(* CoDeSys 2.3.9.41 project: A1.pro *)
(* Libraries: STANDARD.LIB 15.6.21 11:37:35, IECSFC.LIB 15.6.21 11:37:35, SYSLIBTIME.LIB 18.6.21 10:30:26, SYSTASKINFO.LIB 18.6.21 10:30:26, ANALYZATION.LIB 15.6.21 11:37:35, SYSLIBCALLBACK.LIB 18.6.21 10:30:26 *)

(* PLC configuration (modules and I/O channels)
DI_1 AT %IX0.0 [BitInput] Discrete input 1 {ChannellName = Enter name}
DI_2 AT %IX0.1 [BitInput] Discrete input 2 {ChannellName = Enter name}
Discrete inputs [ID130] node 1, in %IB1 out %QB1 {ChannellName = Discrete inputs; Filtrationtime_GeneralINP = 16; PinCount = 16}
  AT %IB1.0 [ByteInput] 8 discrete inputs {ChannellName = Enter name}
  AT %IB1.1 [ByteInput] 8 discrete inputs {ChannellName = Enter name}
DO_1 AT %QX2.0 [BitOutput] Fast discrete output 1 {ChannellName = Enter name}
DO_2 AT %QX2.1 [BitOutput] Fast discrete output 2 {ChannellName = Enter name}
DO_3 AT %QX2.2 [BitOutput] Fast discrete output 3 {ChannellName = Enter name}
DO_4 AT %QX2.3 [BitOutput] Fast discrete output 4 {ChannellName = Enter name}
AT %QB3.0 [ByteOutput] 8 discrete outputs {ChannellName = Enter name}
AT %QB3.1 [ByteOutput] 8 discrete outputs {ChannellName = Enter name}
Special input [ID103] node 4, in %IB4 out %QB4 {ChannellName = Special input}
  AT %IX4.0 [BitInput] Special input {ChannellName = Enter name}
Special output [ID104] node 5, in %IB5 out %QB5 {ChannellName = Special output}
  AT %QX5.0 [BitOutput] Special output {ChannellName = Enter name}
RS-485-1 [COM1_USART] node 0, in %IB6.0.0 out %QB6.0.0 {ChannellName = RS-485-1; CommunicationSpeed = 115200; Parity = NO PARITY CHECK; BitLength = 8 bits; StopLength = One stop bit; InterfaceType = RS485; FrameOriented = RTU; Timeout = 0; Visibility = No}
2 byte [Register] node 1, in %IB6.1 out %QB6.1 {ChannellName = 2 byte}
  DI AT %QW6.1.0 [WordOutput] {ChannellName = Enter name}
2 byte [Register] node 2, in %IB6.2 out %QB6.2 {ChannellName = 2 byte}
  DOMod AT %QW6.2.0 [WordOutput] {ChannellName = Enter name}
2 byte [Register] node 3, in %IB6.3 out %QB6.3 {ChannellName = 2 byte}
  iPressure1 AT %QW6.3.0 [WordOutput] {ChannellName = Enter name}
2 byte [Register] node 4, in %IB6.4 out %QB6.4 {ChannellName = 2 byte}
  iPressure2 AT %QW6.4.0 [WordOutput] {ChannellName = Enter name}
2 byte [Register] node 5, in %IB6.5 out %QB6.5 {ChannellName = 2 byte}
  iPressure3 AT %QW6.5.0 [WordOutput] {ChannellName = Enter name}
2 byte [Register] node 6, in %IB6.6 out %QB6.6 {ChannellName = 2 byte}
  iPressure4 AT %QW6.6.0 [WordOutput] {ChannellName = Enter name}
2 byte [Register] node 7, in %IB6.7 out %QB6.7 {ChannellName = 2 byte}
  iPressure5 AT %QW6.7.0 [WordOutput] {ChannellName = Enter name}
2 byte [Register] node 8, in %IB6.8 out %QB6.8 {ChannellName = 2 byte}
  iPressure6 AT %QW6.8.0 [WordOutput] {ChannellName = Enter name}
2 byte [Register] node 9, in %IB6.9 out %QB6.9 {ChannellName = 2 byte}
  iPressureAll AT %QW6.9.0 [WordOutput] {ChannellName = Enter name}
2 byte [Register] node 10, in %IB6.10 out %QB6.10 {ChannellName = 2 byte}
  iPressureOil AT %QW6.10.0 [WordOutput] {ChannellName = Enter name}
2 byte [Register] node 11, in %IB6.11 out %QB6.11 {ChannellName = 2 byte}
  qNeedTemp AT %QW6.11.0 [WordOutput] {ChannellName = Enter name}
2 byte [Register] node 12, in %IB6.12 out %QB6.12 {ChannellName = 2 byte}
  qTempDelta AT %QW6.12.0 [WordOutput] {ChannellName = Enter name}
2 byte [Register] node 13, in %IB6.13 out %QB6.13 {ChannellName = 2 byte}
  qPressureOilMax AT %QW6.13.0 [WordOutput] {ChannellName = Enter name}
2 byte [Register] node 14, in %IB6.14 out %QB6.14 {ChannellName = 2 byte}
  qPressureMax AT %QW6.14.0 [WordOutput] {ChannellName = Enter name}
2 byte [Register] node 15, in %IB6.15 out %QB6.15 {ChannellName = 2 byte}
  qTempMin AT %QW6.15.0 [WordOutput] {ChannellName = Enter name}
2 byte [Register] node 16, in %IB6.16 out %QB6.16 {ChannellName = 2 byte}
  iAlarms AT %QW6.16.0 [WordOutput] {ChannellName = Enter name}
2 byte [Register] node 17, in %IB6.17 out %QB6.17 {ChannellName = 2 byte}
  qNeedPressure1 AT %QW6.17.0 [WordOutput] {ChannellName = Enter name}
2 byte [Register] node 18, in %IB6.18 out %QB6.18 {ChannellName = 2 byte}
  qNeedPressure2 AT %QW6.18.0 [WordOutput] {ChannellName = Enter name}
2 byte [Register] node 19, in %IB6.19 out %QB6.19 {ChannellName = 2 byte}
  qNeedPressure3 AT %QW6.19.0 [WordOutput] {ChannellName = Enter name}
2 byte [Register] node 20, in %IB6.20 out %QB6.20 {ChannellName = 2 byte}
  qNeedPressure4 AT %QW6.20.0 [WordOutput] {ChannellName = Enter name}
  qNeedPressure5 AT %QW6.21.0 [WordOutput] {ChannellName = Enter name}
  qNeedPressure6 AT %QW6.22.0 [WordOutput] {ChannellName = Enter name}
  iTemp1 AT %QW6.23.0 [WordOutput] {ChannellName = Enter name}
  iTemp2 AT %QW6.24.0 [WordOutput] {ChannellName = Enter name}
  iTemp3 AT %QW6.25.0 [WordOutput] {ChannellName = Enter name}
  iTemp4 AT %QW6.26.0 [WordOutput] {ChannellName = Enter name}
  iTemp5 AT %QW6.27.0 [WordOutput] {ChannellName = Enter name}
  iTemp6 AT %QW6.28.0 [WordOutput] {ChannellName = Enter name}
  qTime1 AT %QW6.29.0 [WordOutput] {ChannellName = Enter name}
  qTime2 AT %QW6.30.0 [WordOutput] {ChannellName = Enter name}
  qTime3 AT %QW6.31.0 [WordOutput] {ChannellName = Enter name}
  qTime4 AT %QW6.32.0 [WordOutput] {ChannellName = Enter name}
  qTime5 AT %QW6.33.0 [WordOutput] {ChannellName = Enter name}
  qTime6 AT %QW6.34.0 [WordOutput] {ChannellName = Enter name}
  iAutoStatus AT %QW6.35.0 [WordOutput] {ChannellName = Enter name}
AT %QD7.0 [DWordOutput] Last address {ChannellName = Enter name}
AT %QW7.1 [WordOutput] Last error {ChannellName = Enter name}
Empty [Empty_module] node 0, in %IB7.0 out %QB7.0 {ChannellName = Empty slot}
AT %QB7.1.0 [ComChannel] Command (0xff - Start) {ChannellName = Enter name}
iNeedTemp AT %QW7.1.0.0 [WordOutput] {ChannellName = Enter name}
qPressure1 AT %QW7.1.1.0 [WordOutput] {ChannellName = Enter name}
qPressure2 AT %QW7.1.2.0 [WordOutput] {ChannellName = Enter name}
qPressure3 AT %QW7.1.3.0 [WordOutput] {ChannellName = Enter name}
qPressure4 AT %QW7.1.4.0 [WordOutput] {ChannellName = Enter name}
qPressure5 AT %QW7.1.5.0 [WordOutput] {ChannellName = Enter name}
qPressure6 AT %QW7.1.6.0 [WordOutput] {ChannellName = Enter name}
iNeedPressure1 AT %QW7.1.7.0 [WordOutput] {ChannellName = Enter name}
iNeedPressure2 AT %QW7.1.8.0 [WordOutput] {ChannellName = Enter name}
iNeedPressure3 AT %QW7.1.9.0 [WordOutput] {ChannellName = Enter name}
iNeedPressure4 AT %QW7.1.10.0 [WordOutput] {ChannellName = Enter name}
iNeedPressure5 AT %QW7.1.11.0 [WordOutput] {ChannellName = Enter name}
iNeedPressure6 AT %QW7.1.12.0 [WordOutput] {ChannellName = Enter name}
qAlarms AT %QW7.1.13.0 [WordOutput] {ChannellName = Enter name}
qTemp1 AT %QW7.1.14.0 [WordOutput] {ChannellName = Enter name}
qTemp2 AT %QW7.1.15.0 [WordOutput] {ChannellName = Enter name}
qTemp3 AT %QW7.1.16.0 [WordOutput] {ChannellName = Enter name}
qTemp4 AT %QW7.1.17.0 [WordOutput] {ChannellName = Enter name}
qTemp5 AT %QW7.1.18.0 [WordOutput] {ChannellName = Enter name}
qTemp6 AT %QW7.1.19.0 [WordOutput] {ChannellName = Enter name}
qPressureAll AT %QW7.1.20.0 [WordOutput] {ChannellName = Enter name}
qPressureOil AT %QW7.1.21.0 [WordOutput] {ChannellName = Enter name}
iTempMin AT %QW7.1.22.0 [WordOutput] {ChannellName = Enter name}
iTempDelta AT %QW7.1.23.0 [WordOutput] {ChannellName = Enter name}
iPressureOilMax AT %QW7.1.24.0 [WordOutput] {ChannellName = Enter name}
iPressureAllMax AT %QW7.1.25.0 [WordOutput] {ChannellName = Enter name}
iTime1 AT %QW7.1.26.0 [WordOutput] {ChannellName = Enter name}
iTime2 AT %QW7.1.27.0 [WordOutput] {ChannellName = Enter name}
iTime3 AT %QW7.1.28.0 [WordOutput] {ChannellName = Enter name}
iTime4 AT %QW7.1.29.0 [WordOutput] {ChannellName = Enter name}
iTime5 AT %QW7.1.30.0 [WordOutput] {ChannellName = Enter name}
iTime6 AT %QW7.1.31.0 [WordOutput] {ChannellName = Enter name}
qAutoStatus AT %QW7.1.32.0 [WordOutput] {ChannellName = Enter name}
*)

(* POU PLC_PRG, ST *)
PROGRAM PLC_PRG
VAR

	(* ВХОДЫ *)
	button1sec1:BOOL;
	button2sec1:BOOL;
	openButtonSec1:BOOL;


	button1sec2:BOOL;
	button2sec2:BOOL;
	openButtonSec2:BOOL;

	button1sec3:BOOL;
	button2sec3:BOOL;
	openButtonSec3:BOOL;

	button1sec4:BOOL;
	button2sec4:BOOL;
	openButtonSec4:BOOL;

	button1sec5:BOOL;
	button2sec5:BOOL;
	openButtonSec5:BOOL;

	button1sec6:BOOL;
	button2sec6:BOOL;
	openButtonSec6:BOOL;


	(* ВЫХОДЫ *)

	AlarmControl:BOOL;

	hydroEngine:BOOL;


	dSec1:BOOL;
	dSec1FB:togetherButtons;
	dSec2:BOOL;
	dSec2FB:togetherButtons;
	dSec3:BOOL;
	dSec3FB:togetherButtons;
	dSec4:BOOL;
	dSec4FB:togetherButtons;
	dSec5:BOOL;
	dSec5FB:togetherButtons;
	dSec6:BOOL;
	dSec6FB:togetherButtons;


END_VAR
button1sec1:=DI_1;
button2sec1:=DI_2;
openButtonSec1:=DI_3;

button1sec2:=DI_4;
button2sec2:=DI_5;
openButtonSec2:=DI_6;

button1sec3:=DI_7;
button2sec3:=DI_8;
openButtonSec3:=DI_9;

button1sec4:=DI_10;
button2sec4:=DI_11;
openButtonSec4:=DI_12;

button1sec5:=DI_13;
button2sec5:=DI_14;
openButtonSec5:=DI_15;

button1sec6:=DI_16;
button2sec6:=DI_17;
openButtonSec6:=DI_18;




DO_13:=AlarmControl;
DO_14:=hydroEngine;

dSec1FB(button1:= button1Sec1, button2:=button2Sec1 , out=>dSec1 );
dSec2FB(button1:= button1Sec2, button2:=button2Sec2 , out=>dSec2 );
dSec3FB(button1:= button1Sec3, button2:=button2Sec3 , out=>dSec3 );
dSec4FB(button1:= button1Sec4, button2:=button2Sec4 , out=>dSec4 );
dSec5FB(button1:= button1Sec5, button2:=button2Sec5 , out=>dSec5 );
dSec6FB(button1:= button1Sec6, button2:=button2Sec6 , out=>dSec6 );

DI.0:=openButtonSec1;
DI.1:=openButtonSec2;
DI.2:=openButtonSec3;
DI.3:=openButtonSec4;
DI.4:=openButtonSec5;
DI.5:=openButtonSec6;
DI.6:=dSec1;
DI.7:=dSec2;
DI.8:=dSec3;
DI.9:=dSec4;
DI.10:=dSec5;
DI.11:=dSec6;
(*
DI.12:=openButtonSec1;
DI.13:=openButtonSec1;
DI.14:=openButtonSec1;
DI.15:=openButtonSec1;
DI.16:=openButtonSec1; 
*)




AlarmControl:=DOMod.12;
hydroEngine:=DOMod.13;

qPressure1:=iPressure1;
qPressure2:=iPressure2;
qPressure3:=iPressure3;
qPressure4:=iPressure4;
qPressure5:=iPressure5;
qPressure6:=iPressure6;
qNeedPressure1:=iNeedPressure1;
qNeedPressure2:=iNeedPressure2;
qNeedPressure3:=iNeedPressure3;
qNeedPressure4:=iNeedPressure4;
qNeedPressure5:=iNeedPressure5;
qNeedPressure6:=iNeedPressure6;

qNeedTemp:=iNeedTemp;
qPressure1:=iPressure1;
qPressure2:=iPressure2;
qPressure3:=iPressure3;
qPressure4:=iPressure4;
qPressure5:=iPressure5;
qPressure6:=iPressure6;
qTemp1:=iTemp1;
qTemp2:=iTemp2;
qTemp3:=iTemp3;
qTemp4:=iTemp4;
qTemp5:=iTemp5;
qTemp6:=iTemp6;


qPressureAll:=iPressureAll;

qPressureOil:=iPressureOil;
qAlarms:=iAlarms;
qTempDelta:=iTempDelta;
qTempMin:=iTempMin;
qTime1:=iTime1;
qTime2:=iTime2;
qTime3:=iTime3;
qTime4:=iTime4;
qTime5:=iTime5;
qTime6:=iTime6;
qAutoStatus:=iAutoStatus;
END_PROGRAM

(* POU togetherButtons, ST *)
FUNCTION_BLOCK togetherButtons
VAR_INPUT
	button1:BOOL;
	button2:BOOL;
END_VAR
VAR_OUTPUT
	out:BOOL;
END_VAR
VAR
	button1Main:BOOL;
	button2Main:BOOL;
	timer1:TP;
	timer2:TP;
	main:SR;
END_VAR
timer1(IN:=button1, PT:=T#255ms , Q=>button1Main);
timer2(IN:=button2, PT:=T#255ms , Q=>button2Main);
main(SET1:= button1Main AND button2Main, RESET:=NOT button1 OR NOT button2, Q1=>out);
END_FUNCTION_BLOCK
